TYPE SStatistic_t :
STRUCT
	u32TestSuites   : UDINT;
	u32TestCases 	: UDINT;
	u32Executed 	: UDINT;
	u32Asserts 		: UDINT;
	u32Passed 		: UDINT;
	u32Failed 		: UDINT;
END_STRUCT
END_TYPE

(* stored: Version 1.1.0.1, ProductVersion 3.1.4022.12
   DUT SStatistic_t: Id {1bab325b-bebc-4938-9dd0-fcf6492717ca} *)
